Fanuc KAREL source: kt00502.KL

-- PROVISIONAL review KL for V1013-1; original PC SHA256 b68f3b76c81e9ee5ced6c88a8bac28527b23567be3944059b97d36d1da32fa68
-- Incomplete behavior may be omitted. Consult companion uncertainty JSON. Do not deploy.
PROGRAM KT00502
%NOLOCKGROUP
-- UNRESOLVED_DECL P1 type=000102
-- UNRESOLVED_DECL P2 type=000102
-- UNRESOLVED_DECL OUT type=000199
BEGIN
  -- UNRESOLVED_PC offsets 5-20; opcodes 2E,22,32,35
  -- UNRESOLVED_PC offsets 25-40; opcodes 2E,22,32,35
  -- UNRESOLVED_PC offsets 45-60; opcodes 2E,22,32,35
  -- UNRESOLVED_PC offsets 65-80; opcodes 2E,22,32,35
  -- UNRESOLVED_PC offsets 85-124; opcodes 49,7E,49,7E,60,7E,4A
  -- UNRESOLVED_PC offsets 129-133; opcodes 7F
END KT00502
